TYPE ST_PDxx_Status :
STRUCT
	bZeroInitialised 			: BOOL := FALSE;
	bReversePolarity			: BOOL;
	nHomePosition				: DINT;
	nCurrentPosition			: DINT;
	nCurrentVelocity			: INT;
	nTargetPosition				: DINT;
	nMinActualPosition			: DINT;
	nMaxActualPosition			: DINT;
	stErrorRegister				: ST_PDxx_ErrorRegister;
	nNumErrors					: USINT;
	ErrorField					: ARRAY [1..8] OF ST_PDxx_PredefinedErrorField;
END_STRUCT
END_TYPE

(* stored: Version 1.1.0.1, ProductVersion 3.1.4024.15
   DUT ST_PDxx_Status: Id {182bda49-5b13-411c-ba43-6b60cb22b1dd} *)
